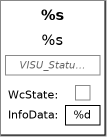
VISUALIZATION VISU_EtherCatDevice  // 107x137
VAR_IN_OUT
	device : EtherCatDevice;
	widget : EtherCatDeviceWidget;
END_VAR
    Rectangle (0,0 105x135)
    Rectangle (0,0 105x30), "%s", text variable: device.typeId
    Rectangle (0,25 105x30), "%s", text variable: device.id
    Label (5,80 60x30), "WcState:"
    Label (5,100 60x30), "InfoData:"
    Rectangle (65,105 35x20), "%d", text variable: device.infoData
    Frame (5,55 95x20)
        shows VISU_StatusWidget(widget := widget.actualStatus)
    Frame (75,85 15x15)
        shows VISU_State_green_red(state := device.wcState)
END_VISUALIZATION

(* stored: Version 1.1.0.1, ProductVersion 3.1.4019.2
   Visu VISU_EtherCatDevice: Id {ecd9b44e-7e4a-498b-be53-7759dfbc2a9b} *)
